{attribute 'qualified_only'}
VAR_GLOBAL

//Block States IO
mInSwitch : ARRAY[0..76] OF DINT;
mOutSwitch : ARRAY[0..76] OF DINT;
mInOccupancies : ARRAY[0..76] OF DINT;
mOutOccupancies : ARRAY[0..76] OF DINT;
mInSpeeds : ARRAY[0..76] OF DINT;
mOutSpeeds : ARRAY[0..76] OF DINT;
mInAuthorities : ARRAY[0..76] OF DINT;
mOutAuthorities : ARRAY[0..76] OF DINT;
mInCrossings : ARRAY[0..76] OF DINT;
mOutCrossings : ARRAY[0..76] OF DINT;
mInLeftLights : ARRAY[0..76] OF DINT;
mOutLeftLights : ARRAY[0..76] OF DINT;
mInRightLights : ARRAY[0..76] OF DINT;
mOutRightLights : ARRAY[0..76] OF DINT;
mInMaintenance : ARRAY[0..76] OF DINT;
mOutMaintenance : ARRAY[0..76] OF DINT;

END_VAR

(* stored: Version 1.1.0.1, ProductVersion 3.1.4024.11
   GVL GVL: Id {e116494b-008e-4148-a200-cfa04c206013} *)
